PROGRAM pouMsgS3
VAR
	
	
	
END_VAR

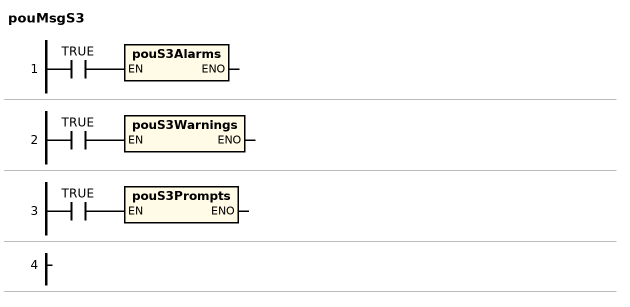
// NETWORK 1
pouS3Alarms();

// NETWORK 2
pouS3Warnings();

// NETWORK 3
pouS3Prompts();

// NETWORK 4

END_PROGRAM

(* stored: Version 1.1.0.1, ProductVersion 3.1.4024.12
   POU pouMsgS3: Id {14de976c-e076-423c-8c07-ae9a846373d9}, SpecialFunc None *)
